INTERFACE I_LWORD EXTENDS I_Datatype

PROPERTY PUBLIC Value : REFERENCE TO LWORD
GET
END_GET
END_PROPERTY

END_INTERFACE

(* stored: Version 1.1.0.1, ProductVersion 3.1.4024.15
   Itf I_LWORD: Id {3ad6bf80-55cc-0b7f-36c3-d0c11f83a142}
   Property Value: Id {59ae7cc2-aa8a-054b-1a6a-bdec2057d45d}
   Get Get: Id {b387d43e-7713-09cc-0e7e-6c1d70312d4e} *)
